Staubli VAL3: buildList.pgx

program buildList()
  local num l_nSize
  local num i
  local string l_sInstruction
  local string l_sMessage
  local string l_sTemp
  local string l_sEmpty
  local string l_sData
  local string l_sType
begin
  call use:setSizeList(13,0,25,9)
  //建立对话款
  call use:listcreate("")
//  l_sEmpty=""
  call use:stringCopy(l_sEmpty,sList)
//  call use:selectNewField(nSelected,nIndex,nView)
  call listAdd("点属性 "+">取片点移动")
  call listAdd("Appro "+" X  > "+toString(".2",data:pPoinTest[data:nPage_Traj].trsf.x))
  call listAdd("Appro "+" Y  > "+toString(".2",data:pPoinTest[data:nPage_Traj].trsf.y))
  call listAdd("Appro "+" Z  > "+toString(".2",data:pPoinTest[data:nPage_Traj].trsf.z))
  call listAdd("Appro "+" RX > "+toString(".2",data:pPoinTest[data:nPage_Traj].trsf.rx))
  call listAdd("Appro "+" RY > "+toString(".2",data:pPoinTest[data:nPage_Traj].trsf.ry))
  call listAdd("Appro "+" RZ > "+toString(".2",data:pPoinTest[data:nPage_Traj].trsf.rz))
  call listAdd("速度 "+" > "+toString(".2",data:mNomSpeed.vel)+"%")
  call listAdd("加速度 "+" > "+toString(".2",data:mNomSpeed.accel)+"%")
  call listAdd("偏移方式  >Appro")
  call listAdd("偏移对象  >摆正点")
  call listAdd("移动方式  >直线")
  call listAdd("停止  >[ ]")
  call listAdd("混合  >[ ]")
  call listAdd("输出提前 > 0mm")
  call use:listadd(sList)
 // nIndex=data:nPage_viewTraj
  call use:selectNewField(nSelected,nIndex,nView)
  call use:listupdate(0)
end
